Yaskawa INFORM job: MASTER_SCIANA_R2.JBI

/JOB
//NAME MASTER_SCIANA_R2
///FOLDERNAME MASTER-SCIANA-R2
//POS
///NPOS 55,55,55,0,0,0
///TOOL 0
///POSTYPE PULSE
///PULSE
C00000=-5011,37072,26260,3759,91732,-85477
C00001=-5011,38780,33406,3752,88219,-85582
C00002=-5012,38778,33409,3767,88218,-85582
C00003=-5011,38780,33406,3752,88219,-85582
C00004=12948,-88986,-121278,-39136,89366,-86840
C00005=13644,-90012,-121559,-38648,88515,-86722
C00006=3049,-150551,-129230,-4221,35623,-81679
C00007=-13512,109275,27441,16100,94054,-76800
C00008=97801,-92951,-68020,42573,91743,-12282
C00009=25883,-65786,-78412,-11285,64556,74084
C00010=-21252,36666,-33912,-7446,103563,-49572
C00011=-147750,-31965,-71698,-11557,98758,-54427
C00012=-28105,107103,24913,6745,88279,-69024
C00013=-1503,48046,-28403,12258,96069,-81953
C00014=4592,-94181,-91931,709,81235,-59832
C00015=-6966,79854,6854,531,84027,-81055
C00016=-29020,140599,41152,11742,95264,-86026
C00017=78395,-65344,-80275,11767,96148,-85942
C00018=-112867,-145355,-130280,83721,-18285,930
C00019=-112867,-145355,-130280,-5739,-2626,930
C00020=-46432,-159370,-130280,-2544,61420,930
C00021=-19143,-90996,-91728,16686,73413,-40961
C00022=-13148,3851,-75147,-6736,62300,-60674
C00023=-42977,-18772,-75159,22659,79337,-61702
C00024=6001,25874,-16138,-19603,78346,75518
C00025=-11894,-51723,-75150,12718,83736,79808
C00026=-11894,-51723,-75150,12718,83736,79808
C00027=-20488,132232,36241,15315,95213,-79268
C00028=19116,-86609,-130129,-2582,74400,63771
C00029=-23133,119915,11793,10868,102368,-84878
C00030=-23133,119915,11793,10868,102368,-84878
C00031=99911,-177915,-134930,-14535,-6478,-4116
C00032=113339,-169627,-129785,-11895,253,-2377
C00033=10051,-169051,-129428,-11712,75776,-2256
C00034=10417,-169879,-125602,29215,16410,-73704
C00035=113735,-122420,-119423,19643,55864,-58497
C00036=113735,-122420,-119423,19643,55864,-58497
C00037=13699,-122420,-119423,19643,55864,-58497
C00038=-9572,-16705,-102894,16661,99188,-59602
C00039=13527,-43767,-75037,30600,77310,-61859
C00040=-3198,-159049,-135849,-2636,-13662,-61972
C00041=16374,-141640,-130183,11627,90903,-81632
C00042=-119308,-141640,-130183,10560,13476,-81264
C00043=-119308,-141640,-130183,10560,13476,-81264
C00044=-176477,-141640,-130183,11345,42887,-77263
C00045=-139275,-147023,-123900,66598,-4025,-48175
C00046=-8798,-147023,-123900,66598,-4025,-48175
C00047=-5748,-152569,-126248,19414,31869,82321
C00048=-5748,-152569,-126248,19414,31869,82321
C00049=-6081,-148304,-123918,19275,32833,80021
C00050=22999,-153190,-124770,8193,30097,64033
C00051=-5011,37072,26260,3759,91732,-85477
C00052=-5210,22770,-28637,-16638,85398,8090
C00053=-5011,38780,33406,3752,88219,-85582
C00054=-5011,38780,33406,3752,88219,-85582
BC00000=62200,671721,936296
BC00001=62200,686065,1044826
BC00002=62201,686062,1044820
BC00003=62200,680360,1044826
BC00004=196190,669163,1073599
BC00005=195682,795553,1072325
BC00006=86842,666865,1035234
BC00007=107345,714512,1049058
BC00008=366006,1114529,810332
BC00009=316850,1266855,846608
BC00010=169338,1219832,1032988
BC00011=338826,1029572,1025585
BC00012=88670,742328,1070144
BC00013=178400,865242,1050786
BC00014=295772,746316,1055266
BC00015=87730,719512,1070892
BC00016=87730,811779,1070892
BC00017=316083,861355,1070892
BC00018=394279,879620,1059380
BC00019=394279,1263974,1059380
BC00020=394279,1263974,1059380
BC00021=345510,1299246,1065426
BC00022=5303,692917,1023031
BC00023=124867,756769,1070853
BC00024=73330,743948,1045976
BC00025=60692,677201,1068222
BC00026=60692,677201,1068222
BC00027=137913,743915,1070893
BC00028=60102,670455,1062776
BC00029=126121,729545,1068204
BC00030=126121,1057038,1068204
BC00031=19015,735315,660782
BC00032=6446,1223776,683902
BC00033=5573,1164495,685508
BC00034=164421,684835,1022347
BC00035=21500,1191142,1068221
BC00036=21500,874764,1068221
BC00037=22298,732932,1068221
BC00038=13731,1269358,1070905
BC00039=86599,727322,1068222
BC00040=25189,722041,1068222
BC00041=107378,765575,1068205
BC00042=255400,765575,1068205
BC00043=386182,939595,1068205
BC00044=370902,1048659,1068205
BC00045=317786,724467,1069775
BC00046=222211,724467,1069775
BC00047=209163,732859,1067793
BC00048=209163,732859,1067793
BC00049=207194,1219066,1066584
BC00050=94818,682102,1068222
BC00051=62200,671721,936296
BC00052=125677,684263,1067629
BC00053=62200,686065,1044826
BC00054=62200,686065,809464
EC00000=0,556475
EC00001=0,556475
EC00002=-830412,0
EC00003=0,556475
EC00004=798152,2
EC00005=798147,2
EC00006=798150,2
EC00007=0,556476
EC00008=0,556476
EC00009=0,556476
EC00010=1,556476
EC00011=1,556476
EC00012=1,556476
EC00013=1,556476
EC00014=-371563,-8038
EC00015=1,556476
EC00016=1,556476
EC00017=1,556476
EC00018=-798157,556476
EC00019=-798157,556476
EC00020=-798157,556476
EC00021=-798156,556476
EC00022=-798157,1112952
EC00023=620788,1112951
EC00024=798153,1112951
EC00025=399078,1112952
EC00026=0,1112952
EC00027=0,556476
EC00028=-709464,556478
EC00029=-798157,0
EC00030=-798157,0
EC00031=-798157,-556476
EC00032=-798157,-556476
EC00033=-798157,-556476
EC00034=-798152,-556475
EC00035=-798150,-556477
EC00036=-798150,-556477
EC00037=-798150,-556477
EC00038=-798150,-556477
EC00039=-709473,-556476
EC00040=-1596314,556476
EC00041=-1596314,556476
EC00042=-1596314,556476
EC00043=-1596314,556476
EC00044=-1596314,556476
EC00045=-1596313,556476
EC00046=-1596313,556476
EC00047=-1596314,-556476
EC00048=-1596314,-556476
EC00049=-1152894,1112952
EC00050=-1064209,1112952
EC00051=0,556475
EC00052=-923702,-5089
EC00053=0,556475
EC00054=0,556475
//INST
///DATE 2024/07/30 13:24
///ATTR SC,RW
///GROUP1 RB1,BS1
///GROUP2 ST1
NOP
MOVJ C00000 BC00000 VJ=100.00  +MOVJ EC00000 VJ=100.00
MOVJ C00001 BC00001 VJ=100.00  +MOVJ EC00001 VJ=100.00
MOVJ C00002 BC00002 VJ=100.00  +MOVJ EC00002 VJ=100.00
PAUSE
PAUSE
'UWAGA!!!!
'SCIAGNAC UCHWYTY SCIANY
MOVJ C00003 BC00003 VJ=100.00  +MOVJ EC00003 VJ=100.00
CALL JOB:0_-90
CALL JOB:R1_W01(KAMERA)(0,-90)NEW
CALL JOB:125_90
CALL JOB:R1_W12(125,90)(KAMERA)
CALL JOB:-90_90
CALL JOB:R1_W26(-90,90)(KAMERA)
COMM CALL JOB:R1_W26(-90,90)(KAMERA)
CALL JOB:R1_W23(-90,90)(KAMERA)KM-OK
MOVJ C00004 BC00004 VJ=100.00  +MOVJ EC00004 VJ=40.00
CALL JOB:R1_W24(-90,90)KM-OK
MOVJ C00005 BC00005 VJ=100.00  +MOVJ EC00005 VJ=100.00
MOVJ C00006 BC00006 VJ=100.00  +MOVJ EC00006 VJ=100.00
'KONIEC SPAWANIA ZE SLEDZENIEM
'KAMERA SERVO ROBOT
'----------------------
CALL JOB:ONLY_CUT_KM_NEW_SCIANA
CALL JOB:0_0
MOVJ C00007 BC00007 VJ=100.00  +MOVJ EC00007 VJ=30.00
MOVJ C00008 BC00008 VJ=100.00  +MOVJ EC00008 VJ=40.00
CALL JOB:R1_W03,5,7(0,0)OK-KM
CALL JOB:ONLY_CUT_KM_NEW_SCIANA
MOVJ C00009 BC00009 VJ=100.00  +MOVJ EC00009 VJ=100.00
MOVJ C00010 BC00010 VJ=100.00  +MOVJ EC00010 VJ=40.00
MOVJ C00011 BC00011 VJ=100.00  +MOVJ EC00011 VJ=40.00
CALL JOB:R1_W02,4,6(0_0)_KM-OK
MOVJ C00012 BC00012 VJ=100.00  +MOVJ EC00012 VJ=100.00
CALL JOB:CLEAN-R1_KM_NEW_SCIANA
CALL JOB:R1_W14,16(0,0)OK-KM
CALL JOB:CLEAN-R1_KM_NEW_SCIANA
CALL JOB:R1_W13,15(0,0)KM-OK
CALL JOB:ONLY_CUT_KM_NEW_SCIANA
MOVJ C00013 BC00013 VJ=100.00  +MOVJ EC00013 VJ=100.00
MOVJ C00014 BC00014 VJ=99.00  +MOVJ EC00014 VJ=99.00
CALL JOB:R1_W17,20,22(0,0)OK-KMNEW2
MOVJ C00015 BC00015 VJ=40.00  +MOVJ EC00015 VJ=25.00
CALL JOB:CLEAN-R1_KM_NEW_SCIANA
MOVJ C00016 BC00016 VJ=40.00  +MOVJ EC00016 VJ=40.00
MOVJ C00017 BC00017 VJ=40.00  +MOVJ EC00017 VJ=40.00
'DODANE SEARCH
CALL JOB:R1_W18,19,21(0,0)_KM-OKNEW_MP
CALL JOB:CLEAN-R1_KM_NEW_SCIANA
CALL JOB:R1_W30(0,0)OK-KM
CALL JOB:ONLY_CUT_KM_NEW_SCIANA
CALL JOB:R1_W33(0,0)KM-OK
CALL JOB:CLEAN-R1_KM_NEW_SCIANA
CALL JOB:R1_W31(0,0)_KM-OK
'----------------------
'SPAWANIE DLA POZYCJI 90_0
CALL JOB:90_0
MOVJ C00018 BC00018 VJ=100.00  +MOVJ EC00018 VJ=100.00
MOVJ C00019 BC00019 VJ=100.00  +MOVJ EC00019 VJ=100.00
MOVJ C00020 BC00020 VJ=100.00  +MOVJ EC00020 VJ=100.00
MOVJ C00021 BC00021 VJ=100.00  +MOVJ EC00021 VJ=40.00
CALL JOB:CLEAN-R1_KM_NEW_SCIANA
CALL JOB:R1_W27-A3(90,0)OK-KM
CALL JOB:ONLY_CUT_KM_NEW_SCIANA
CALL JOB:R1_W27-A5(90,0)OK-KM
CALL JOB:CLEAN-R1_KM_NEW_SCIANA
CALL JOB:R1_W35-36-A2(90,0)KM-OK
CALL JOB:ONLY_CUT_KM_NEW_SCIANA
CALL JOB:R1_W45-48(90,0)KM-OK
'W39-53
CALL JOB:R1_W39(90,0)R2
'---------------------
'SPAWANIE DLA POZYCJI 90_-90
CALL JOB:90_-90
MOVJ C00022 BC00022 VJ=100.00  +MOVJ EC00022 VJ=100.00
CALL JOB:CLEAN-R1_KM_NEW_SCIANA
CALL JOB:R1_W27-A2(90,-90)POPR-KM-OK
CALL JOB:CLEAN-R1_KM_NEW_SCIANA
CALL JOB:R1_W29-KM-NOWY-MP
'---------------------
'ZMIANA POZYCJI SPAWANIA -70_-90
'AWOK
CALL JOB:-70_-90
MOVJ C00023 BC00023 VJ=100.00  +MOVJ EC00023 VJ=40.00
CALL JOB:CLEAN-R1_KM_NEW_SCIANA
CALL JOB:R1_W09,10(-70,-90)
CALL JOB:ONLY_CUT_KM_NEW_SCIANA
CALL JOB:R1_W08,11(-70,-90)_KM-OK
CALL JOB:ONLY_CUT_KM_NEW_SCIANA
CALL JOB:R1_W66-67(-70,-90)KM-OK
CALL JOB:ONLY_CUT_KM_NEW_SCIANA
CALL JOB:R1_W66-W67(-70,-90)KM-OK
'---------------------
'AWOK
'ZMIANA POZYCJI SPAWANIA -90_-90
CALL JOB:-90_-90
CALL JOB:ONLY_CUT_KM_NEW_SCIANA
CALL JOB:R1_W68-69(-90,-90)KM-OK
CALL JOB:CLEAN-R1_KM_NEW_SCIANA
CALL JOB:R1_W68-69(-90,-90)KM-OK-R2
CALL JOB:ONLY_CUT_KM_NEW_SCIANA
CALL JOB:R1_W70(-90,-90)KM-OK
MOVJ C00024 BC00024 VJ=100.00  +MOVJ EC00024 VJ=100.00
'ZMIANA POZYCJI SPAWANIA -45_-90
CALL JOB:-45_-90
CALL JOB:CLEAN-R1_KM_NEW_SCIANA
CALL JOB:R1_W72(-45,-90)KM-OK
CALL JOB:CLEAN-R1_KM_NEW_SCIANA
CALL JOB:R1_W72(-45,-90)R2
MOVJ C00025 BC00025 VJ=100.00  +MOVJ EC00025 VJ=100.00
'ZMIANA POZYCJI SPAWANIA 0_-90
CALL JOB:0_-90
MOVJ C00026 BC00026 VJ=100.00  +MOVJ EC00026 VJ=30.00
CALL JOB:ONLY_CUT_KM_NEW_SCIANA
CALL JOB:R1_W73(0,-90)KM-OK
'ZMIANA POZYCJI SPAWANIA 0_0
'AWOK
MOVJ C00027 BC00027 VJ=100.00  +MOVJ EC00027 VJ=100.00
CALL JOB:ONLY_CUT_KM_NEW_SCIANA
CALL JOB:R1_72,2(0,0)KM-OK
CALL JOB:ONLY_CUT_KM_NEW_SCIANA
CALL JOB:R1_72,2(0,0)R2
'ZMIANA POZYCJI SPAWANIA 80_0
CALL JOB:80_0
CALL JOB:CLEAN-R1_KM_NEW_SCIANA
CALL JOB:R1_W43-44-A1(80,0))KM-OK
'ZMIANA POZYCJI SPAWANIA 90_90
MOVJ C00028 BC00028 VJ=100.00  +MOVJ EC00028 VJ=30.00
CALL JOB:CLEAN-R1_KM_NEW_SCIANA
MOVJ C00029 BC00029 VJ=100.00  +MOVJ EC00029 VJ=100.00
MOVJ C00030 BC00030 VJ=100.00  +MOVJ EC00030 VJ=15.00
CALL JOB:R1_W49-52-A2(90,90)KM-OK
CALL JOB:ONLY_CUT_KM_NEW_SCIANA
CALL JOB:R1_W53-A2(90,90)
'ZMIANA POZYCJI SPAWANIA 90_180
CALL JOB:90_180
CALL JOB:CLEAN-R1_KM_NEW_SCIANA
MOVJ C00031 BC00031 VJ=100.00  +MOVJ EC00031 VJ=100.00
MOVJ C00032 BC00032 VJ=100.00  +MOVJ EC00032 VJ=100.00
MOVJ C00033 BC00033 VJ=100.00  +MOVJ EC00033 VJ=100.00
CALL JOB:R1_W27-A4(90,180)KM-OK
SFTOF
MOVJ C00034 BC00034 VJ=100.00  +MOVJ EC00034 VJ=100.00
CALL JOB:ONLY_CUT_KM_NEW_SCIANA
CALL JOB:R1_W35-36-A1(90,180)KM-OK
MOVJ C00035 BC00035 VJ=80.00  +MOVJ EC00035 VJ=0.78
MOVJ C00036 BC00036 VJ=80.00  +MOVJ EC00036 VJ=80.00
MOVJ C00037 BC00037 VJ=80.00  +MOVJ EC00037 VJ=80.00
COMM MOVJ C00038 BC00038 VJ=100.00  +MOVJ EC00038 VJ=10.00
'SPR PRZEJAZDY
CALL JOB:CLEAN-R1_KM_NEW_SCIANA
CALL JOB:R1_W49-52-A1(90,180)KM-OK
CALL JOB:ONLY_CUT_KM_NEW_SCIANA
CALL JOB:R1_W27-A4(90,180)_KM_OKR2
CALL JOB:ONLY_CUT_KM_NEW_SCIANA
CALL JOB:R1_W53-A1(90,180)R2
'ZMIANA POZYCJI SPAWANIA 80_180
CALL JOB:80_180
CALL JOB:CLEAN-R1_KM_NEW_SCIANA
MOVJ C00039 BC00039 VJ=40.00  +MOVJ EC00039 VJ=40.00
CALL JOB:R1_W43-44-A2(80,180)KM-OK
'ZMIANA POZYCJI SPAWANIA 180_0
CALL JOB:180_0
MOVJ C00040 BC00040 VJ=100.00  +MOVJ EC00040 VJ=40.00
CALL JOB:ONLY_CUT_KM_NEW_SCIANA
MOVJ C00041 BC00041 VJ=100.00  +MOVJ EC00041 VJ=100.00
MOVJ C00042 BC00042 VJ=100.00  +MOVJ EC00042 VJ=100.00
MOVJ C00043 BC00043 VJ=100.00  +MOVJ EC00043 VJ=100.00
MOVJ C00044 BC00044 VJ=100.00  +MOVJ EC00044 VJ=100.00
CALL JOB:R1_W49-52-A5(180,0)KM-OK
MOVJ C00045 BC00045 VJ=100.00  +MOVJ EC00045 VJ=20.00
MOVJ C00046 BC00046 VJ=100.00  +MOVJ EC00046 VJ=100.00
CALL JOB:CLEAN-R1_KM_NEW_SCIANA
CALL JOB:R1_W53-A5(180,0)KM-OK_R2
'ZMIANA POZYCJI SPAWANIA 180_180
MOVJ C00047 BC00047 VJ=100.00  +MOVJ EC00047 VJ=100.00
CALL JOB:CLEAN-R1_KM_NEW_SCIANA
MOVJ C00048 BC00048 VJ=40.00  +MOVJ EC00048 VJ=100.00
'ZMIANA POZYCJI SPAWANIA 130_-90
CALL JOB:130_-90
MOVJ C00049 BC00049 VJ=100.00  +MOVJ EC00049 VJ=100.00
CALL JOB:R1_W63-A2(130,-90)(JEDENR)KM-OK
'ZMIANA POZYCJI SPAWANIA 120_-90
CALL JOB:120_-90
CALL JOB:CLEAN-R1_KM_NEW_SCIANA
CALL JOB:R1_W63-A1(120,-90)KM-OK
MOVJ C00050 BC00050 VJ=100.00  +MOVJ EC00050 VJ=50.00
CALL JOB:CLEAN-R1_KM_NEW_SCIANA
CALL JOB:R1_W63-A1(120,-90)KM-OK_R2
CALL JOB:0_0
MOVJ C00051 BC00051 VJ=100.00  +MOVJ EC00051 VJ=100.00
PAUSE
PAUSE
PAUSE
COMM MOVJ C00052 BC00052 VJ=100.00  +MOVJ EC00052 VJ=100.00
COMM PAUSE
COMM 'UWAGA!!!!
COMM 'ZALOZ UCHYWTY DO SCIANY
COMM CALL JOB:0_0
COMM MOVJ C00053 BC00053 VJ=100.00  +MOVJ EC00053 VJ=0.78
COMM MOVJ C00054 BC00054 VJ=100.00  +MOVJ EC00054 VJ=100.00
SFTOF
END
